Staubli VAL3: prgm1.pgx

program prgm1()
begin
  co_x = 20
  co_y = -20
  movel(appro(pPointRx,{co_x,co_y,0,0,0,0}), tTool, mNomSpeed)
  waitEndMove()

end
